SUBAPPLICATION Uebung_071 (* WBSD auf UT ausgeben, Q1 Schalten wenn Speed >0 *)
  (* Standard: 61499-2; Description: Copyright (c) 2023 Meisterschulen am Ostbahnhof This program and the accompanying materials are made available under the terms of the Eclipse Public License 2.0 which is available at https://www.eclipse.org/legal/epl-2.0/ SPDX-License-Identifier: EPL-2.0 *)
  (* Version 1.0, 2023-10-23, Franz Höpfinger, Meisterschulen am Ostbahnhof *)
  IMPORT logiBUS::io::DI::logiBUS_DI;
  IMPORT logiBUS::io::DQ::logiBUS_DO;
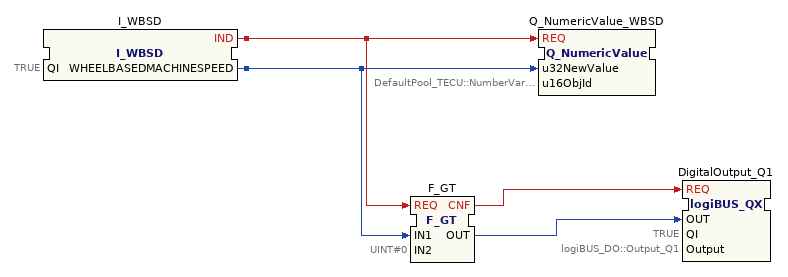
  FBS
    I_WBSD : I_WBSD(QI := TRUE);
    Q_NumericValue_WBSD : isobus::ut::Q_NumericValue(u16ObjId := DefaultPool_TECU::NumberVariable_Wheel_based_machine_speed);
    DigitalOutput_Q1 : logiBUS::io::DQ::logiBUS_QX(QI := TRUE, Output := logiBUS_DO::Output_Q1);
    F_GT : F_GT(IN2 := UINT#0);
  END_FBS
  EVENT_CONNECTIONS
    I_WBSD.IND TO Q_NumericValue_WBSD.REQ;
    I_WBSD.IND TO F_GT.REQ;
    F_GT.CNF TO DigitalOutput_Q1.REQ;
  END_CONNECTIONS
  DATA_CONNECTIONS
    I_WBSD.WHEELBASEDMACHINESPEED TO Q_NumericValue_WBSD.u32NewValue;
    I_WBSD.WHEELBASEDMACHINESPEED TO F_GT.IN1;
    F_GT.OUT TO DigitalOutput_Q1.OUT;
  END_CONNECTIONS
END_SUBAPPLICATION
